// Mitsubishi GX Works2 project: X25   PLC: FX3G

// task Task_01 (event TRUE, interval 0, priority 31): POU_01

PROGRAM POU_01
VAR
  wstep : INT;
  ton1 : TON;
END_VAR
M99 := FALSE AND
M0 AND M1 AND M2 AND
Y0 AND Y1 AND Y2 AND 
Y3 AND Y4 AND Y5;

IF M8002 THEN
	wstep := 0;
END_IF;

IF M2 THEN
	wstep := 100;
END_IF;

CASE wstep OF 
    0:
        zrst(TRUE, Y0, Y5);
        ton1(in := FALSE);

        IF M0 THEN 
            wstep := 20;
        END_IF;
        IF M1 THEN
            wstep := 40;
        END_IF;
    
    20:
        Y5 := TRUE;
        ton1(in := NOT ton1.q, pt := t#5s);
        
        IF ton1.q THEN
            wstep := 21;
        END_IF;
    21:
        Y1 := TRUE;
        Y5 := FALSE;
        ton1(in := NOT ton1.q, pt := t#5s);

        IF ton1.q THEN
            wstep := 22; 
        END_IF;
    22:
        Y0 := TRUE;
        Y1 := FALSE;
        M0 := FALSE;
        ton1(in := NOT ton1.q, pt := t#5s);
        
        IF ton1.q THEN
            wstep := 0;
        END_IF;

    40:
        Y4 := TRUE;
        ton1(in := NOT ton1.q, pt := t#5s);

        IF ton1.q THEN
            wstep := 41;
        END_IF;
    41:
        Y3 := TRUE;
        Y4 := FALSE;
        ton1(in := NOT ton1.q, pt := t#5s);

        IF ton1.q THEN
            wstep := 42;
        END_IF;
    42:
        Y2 := TRUE;
        Y3 := FALSE;
        M1 := FALSE;
        ton1(in := NOT ton1.q, pt := t#5s);

        IF ton1.q THEN
            wstep := 0;
        END_IF;

    100:
        zrst(TRUE, M0, M1);
        zrst(TRUE, Y0, Y5);

        IF NOT M2 THEN
            wstep := 0;
        END_IF;

END_CASE;
END_PROGRAM
